(* IEC 61131-3 sources: crb-codesys/retrieval/output/codesys_repo/轴控/FB101_功能块/F02_模拟滤波, 4 files *)

(* ---- Fun_模拟量比例换算.st ---- *)
FUNCTION Fun_模拟量比例换算 : INT
VAR_INPUT
rOutput: REAL; (* [] Physical output *)
rPhyMin: REAL; (* [] Physical minimum *)
rPhyMax: REAL; (* [] Physical maximum *)
eTerminal: E_Ctrl_TerminalType; (* [] Terminal type. *)
END_VAR
VAR
rTerMin: REAL;
rTerMax: REAL;
rPhyRange: REAL;
rTerRange: REAL;
rTerOutput: REAL;
END_VAR

rTerMax:= 32768.0;

CASE eTerminal OF
eTerminal_0mA_20mA: rTerMin:= 0.0;
eTerminal_4mA_20mA: rTerMin:= 0.0;
eTerminal_0V_10V: rTerMin:= 0.0;
eTerminal_m10V_10V: rTerMin:= -32768.0;
ELSE
rTerMin:= -32768.0;
END_CASE

rPhyRange:= rPhyMax - rPhyMin;
rTerRange:= rTerMax - rTerMin;

IF rPhyRange > 0.0 AND rTerRange > 0.0 THEN
	rTerOutput:= rTerMin + (rTerRange * (rOutput - rPhyMin) / rPhyRange);
ELSE
    rTerOutput:= 0.0;
END_IF

Fun_模拟量比例换算:= REAL_TO_INT(rTerOutput);

(* ---- FB_一阶滤波.st ---- *)
FUNCTION_BLOCK FB_一阶滤波
VAR_INPUT
rInput: REAL:= 0.0; //输入数据
rK: REAL:= 1.0; //增益
tT: TIME; //时间参数
END_VAR
VAR_OUTPUT
rOutput: REAL:= 0.0; //输出数据
END_VAR
VAR
_rT: LREAL;
_rY: LREAL;
END_VAR

IF _rT = 0.0 THEN
    rOutput:= rInput; //输出数据初始化
END_IF
_rT:= TIME_TO_REAL(tT) /10; //10 为 PLC 的采样周期， 单位为 ms

IF ABS(rOutput - rInput) < 1E-6 THEN
    rOutput:= rInput; //防止除零
ELSIF _rT > 0.0 THEN
    rOutput:= (rK / _rT) * rInput + (1.0 - (1.0 / _rT)) * _rY;
ELSE
    rOutput:= rInput; //如果时间常数小于等于零请输出等于输入
END_IF

_rY:= rOutput;

(* ---- FB_模拟量采集滤波.st ---- *)
FUNCTION_BLOCK FB_模拟量采集滤波
VAR_INPUT
    tSampleTime:TIME:=T#200MS; //采样时间
    rInputValue:REAL; //输入数据
END_VAR

VAR_OUTPUT
    rOutputValue:REAL; //输出数据
END_VAR

VAR
    arrBufferData:ARRAY [0..4] OF REAL; //缓存数据
    i:BYTE;
    OverallValue:LREAL;
    fb_SampleTimer:ton;
END_VAR

fb_SampleTimer(IN:= NOT fb_SampleTimer.Q , PT:= tSampleTime);
IF i<5 THEN
   arrBufferData[i]:=rInputValue;
   i:=i+1;
   OverallValue:=arrBufferData[0]+arrBufferData[1]+arrBufferData[2]+arrBufferData[3]+arrBufferData[4];
ELSE
   i:=0;
END_IF

IF fb_SampleTimer.Q THEN
   rOutputValue:=LREAL_TO_REAL(OverallValue/5);
END_IF

(* ---- FB_比例换算.st ---- *)
FUNCTION_BLOCK FB_比例换算
VAR_INPUT
   rIn   :REAL;
   rInMin  :REAL;
   rInMax  :REAL;
   rOutMin  :REAL;
   rOutMax  :REAL;
END_VAR
VAR_OUTPUT
   rOut   :REAL;
END_VAR
VAR
   rK: REAL;
END_VAR

IF rInMax-rInMin<>0  THEN
    rK:=(rOutMax-rOutMin)/(rInMax-rInMin);
END_IF

rOut:=rOutMin+(rIn-rInMin)*rK;
